(* CODESYS project Mbc_Tc3_Pcs.library
   Author: mbc engineering GmbH
   Placeholder: MBC TC3 PCS Library
   Title: MBC TC3 PCS Library
   Version: 1.0.0.0
   DocFormat: reStructuredText
   DefaultNamespace: Mbc_Tc3_Pcs
   Company: mbc engineering GmbH

Project tree, tasks and I/O mapping:
  Command/
    function block CommandBase [ST]: Abort, CalculateProgress, Done, Refresh, Task
    data type E_CommandResultCode
    interface ICommand: Refresh
    data type ST_CommandBaseHandshake
  Version/
    global variables Global_Version
  Mbc_Tc3_Pcs.tmc
  global variables Readme
*)

// Command/E_CommandResultCode
{attribute 'qualified_only'}
{attribute 'strict'}
TYPE E_CommandResultCode :
(
	Init := 0,
	Running := 1,
	Done := 2,
	Cancelled := 3
) UINT;
END_TYPE

// Command/ST_CommandBaseHandshake
TYPE ST_CommandBaseHandshake :
STRUCT
	bExecute		: BOOL;		// Will be set to true from the PCS to start the command. When the operation are finish, the PLC will set the to false. On a long running Task, the PCS can reset to false for Abort the operation. 
	bBusy			: BOOL;		// When the operation is running. Only for multible cycle operations.
	nResultCode		: UINT;		// Shows the operation result code of the commando state. Default Values see 'CommandResultCode' Enum Type.
	nProgress		: UINT;		// Shows the optional calculated progress. The value is depend on the button implementation. (default can be 0..100%). Only necessary on long running operations.
END_STRUCT
END_TYPE

// Version/Global_Version
{attribute 'TcGenerated'}
// This function has been automatically generated from the project information.
VAR_GLOBAL CONSTANT
	{attribute 'const_non_replaced'}
	{attribute 'linkalways'}
	stLibVersion_MBC_TC3_PCS_Library : ST_LibVersion := (iMajor := 1, iMinor := 0, iBuild := 0, iRevision := 0, sVersion := '1.0.0.0');
END_VAR

// Readme
(* 
=================================================
Documentation of mbc engineering GmbH PCS Library
=================================================

:Author: mbc engineering GmbH (MiHe)
:Date: 17.04.2018

This Library will help you to Interagte with the Process Control System (PCS) of mbc engineering GmbH. There are some default exchange logic and structures for reuse. This Library will help you on PLC side on some point. Example on handling PCS commands,

Add the Library Reference
=========================

TBD!

Kick Start with a Command
=========================

First Add a new POU for the Command that extends the Library Class ``CommandBase``.

:Name: 						StartCommand
:Function Block: 			Extends ``CommandBase``
:Access specifier: 			public
:Implementation language: 	at you own decision

Basicly you have a working command that does nothing importand. So we add a Output Parameter.

.. code::
	FUNCTION_BLOCK PUBLIC StartCommand EXTENDS CommandBase
	VAR_INPUT
	END_VAR
	VAR_OUTPUT	
		Q : BOOL;
	END_VAR
	VAR
	END_VAR 

test *)
{attribute 'qualified_only'}
VAR_GLOBAL	
    readme	: ST_LibVersion	:= stLibVersion_MBC_TC3_PCS_Library;  // go to documentation tab
END_VAR

// Command/CommandBase
FUNCTION_BLOCK PUBLIC CommandBase IMPLEMENTS ICommand
VAR_IN_OUT
	(* Use Class Properties for IN_OUT Parameters!!! *)
END_VAR
VAR PERSISTENT
	stHandshake		: ST_CommandBaseHandshake;		// Variable Strukture for communication with PCS. Aditional IN and OUT parameters should be declared in the derived implementation.
END_VAR

// OO-Class 
;

// Stops execution of Command 
METHOD PUBLIC Abort
stHandshake.nResultCode := E_CommandResultCode.Cancelled;
stHandshake.bExecute := FALSE;
stHandshake.bBusy := FALSE;
END_METHOD

METHOD PROTECTED CalculateProgress
IF stHandshake.nResultCode = E_CommandResultCode.Done THEN
	stHandshake.nProgress := 100;
ELSE
	stHandshake.nProgress := 0;
END_IF
END_METHOD

METHOD PROTECTED Done
stHandshake.nResultCode := E_CommandResultCode.Done;
stHandshake.bExecute := FALSE;
stHandshake.bBusy := FALSE;
END_METHOD

// Update the state of the command button. Should be called every cycle.
METHOD PUBLIC Refresh
VAR
	bInit		: BOOL;
END_VAR
// Starting Case
stHandshake.bBusy S= bInit := stHandshake.bExecute AND NOT stHandshake.bBusy;

// Reset Case
IF NOT stHandshake.bExecute AND stHandshake.bBusy THEN
	Abort();
END_IF

// Running Case
IF stHandshake.bExecute AND stHandshake.bBusy THEN
	IF bInit THEN
		stHandshake.nResultCode := E_CommandResultCode.Running;
	END_IF
	
	// Set Task init on First Call
	IF Task(bInit) THEN
		Done();
	END_IF
	
	CalculateProgress();
END_IF
END_METHOD

// Execute the funktional part of the command implementation
METHOD PROTECTED Task : BOOL
VAR_INPUT
	Init 	: BOOL;		// True the first time the Task is called after Execute is started
END_VAR
// Task complete if return true
Task := TRUE;
END_METHOD

END_FUNCTION_BLOCK

// Command/ICommand
INTERFACE ICommand

METHOD Refresh
END_METHOD

END_INTERFACE
